// TwinCAT 3 PLC project PlcIotHttpSamplesOpenWeatherMap
// ProgramVersion: 3.1.4023.0
// libraries:
//   Tc2_Standard, * (Beckhoff Automation GmbH)
//   Tc2_System, * (Beckhoff Automation GmbH)
//   Tc2_Utilities, * (Beckhoff Automation GmbH)
//   Tc3_IotBase, * (Beckhoff Automation GmbH)
//   Tc3_JsonXml, * (Beckhoff Automation GmbH)
//   Tc3_Module, * (Beckhoff Automation GmbH)
// project tree:
//   / PlcTask.TcTTO
//   POUs/ MAIN.TcPOU
//   POUs/OpenWeatherMap/ FB_TestHTTP_Get_openWeatherMap.TcPOU
// (motion and I/O tree: see PLC project plciothttpsamplespostman)
// real-time tasks:
//   TASK PlcTask: cycle T#10ms, priority 20, ADS port 350
//   TASK PlcTask1: cycle T#10ms, priority 21, ADS port 351
//   TASK PlcTask2: cycle T#10ms, priority 22, ADS port 352
//   TASK PlcTask3: cycle T#10ms, priority 23, ADS port 353
//   TASK PlcTask4: cycle T#10ms, priority 24, ADS port 354
//   TASK PlcTask5: cycle T#10ms, priority 25, ADS port 355
//   TASK PlcTask6: cycle T#10ms, priority 26, ADS port 356

CONFIGURATION PlcIotHttpSamplesOpenWeatherMap
    RESOURCE PLC ON TwinCAT3
        TASK PlcTask(INTERVAL := T#10ms, PRIORITY := 23);
        PROGRAM MAIN WITH PlcTask : MAIN;
    END_RESOURCE
END_CONFIGURATION

// ---- POUs/MAIN.TcPOU
PROGRAM MAIN
VAR
	// trigger command execution for OpenWeatherMap samples 	
	bGetOpenWeatherMap 				: BOOL; 

	fbHttpClientOpenWeatherMap		: FB_IotHttpClient :=(sHostName:='api.openweathermap.org',
								  	bKeepAlive:=TRUE,	tConnectionTimeout:=T#10S);

	fbHttpGetOpenWeatherMap			: FB_TestHTTP_Get_openWeatherMap;
END_VAR

// init client parameters at startup
IF NOT fbHttpClientOpenWeatherMap.bConfigured THEN 
	fbHttpClientOpenWeatherMap.nHostPort:= 443;
	fbHttpClientOpenWeatherMap.stTLS.bNoServerCertCheck:= TRUE;
END_IF

IF fbHttpClientOpenWeatherMap.bConfigured THEN
 	fbHttpGetOpenWeatherMap(bSend:=bGetOpenWeatherMap, fbClient:=fbHttpClientOpenWeatherMap);
END_IF

fbHttpClientOpenWeatherMap.Execute();

END_PROGRAM

// ---- POUs/OpenWeatherMap/FB_TestHTTP_Get_openWeatherMap.TcPOU
FUNCTION_BLOCK FB_TestHTTP_Get_openWeatherMap
VAR_INPUT
	bSend				: BOOL;
END_VAR
VAR_IN_OUT
	fbClient			: FB_IotHttpClient;
END_VAR
VAR_OUTPUT
	bBusy				: BOOL;
	bError				: BOOL;
END_VAR
VAR
	fbRequest			: FB_IotHttpRequest;
	fbJson				: FB_JsonDomParser;
	nState				: UDINT;
	RisingEdge			: R_TRIG;
	
	bGetContentResult	: BOOL;
	sContent			: STRING(511);	
	
	bGetJsonResult		: BOOL;
	jsonDoc				: SJsonValue;
	jsonVal				: SJsonValue;
	sResultValue		: STRING;
	
	nReqCount			: UDINT;	
	nResCount			: UDINT;
	nValidResCount		: UDINT;
	nErrCount			: UDINT;
END_VAR

RisingEdge(CLK:= bSend);
CASE nState OF
0:	
	IF RisingEdge.Q THEN 
		IF fbRequest.SendRequest(sUri:='/data/2.5/weather?lat=51.88&lon=8.47&APPID=9adc7censored57f6873e39d', fbClient:=fbClient, eRequestType:=ETcIotHttpRequestType.HTTP_Get, 0, 0, 0) THEN				
			nState:= 1;
			nReqCount:= nReqCount+1;
			bBusy:= TRUE;
			bError:= FALSE;
		END_IF					
	END_IF
1:
	IF NOT fbRequest.bBusy THEN
		bError:= TRUE;
		IF NOT fbRequest.bError THEN				 
			bGetContentResult:= fbRequest.GetContent(pContent:= ADR(sContent), nContentSize:= SIZEOF(sContent), bSetNullTermination:= TRUE);
			IF fbRequest.nStatusCode >= 200 AND fbRequest.nStatusCode < 300 THEN
				bGetJsonResult:= FALSE;
				jsonDoc:= fbRequest.GetJsonDomContent(fbJson);
				IF jsonDoc <> 0 THEN
					; // do something with the weather data
					nValidResCount:= nValidResCount+1;
					bError:= FALSE;					
				END_IF							
				nResCount:= nResCount+1;			
			END_IF
		END_IF
		nState:= 0;
		bBusy:= FALSE;
		IF bError THEN
			nErrCount:= nErrCount+1;
		END_IF
	END_IF  	
END_CASE

END_FUNCTION_BLOCK
